(* IEC 61131-3 sources: Automation-Studio-Files/, 2 files *)

(* ---- Global.var ---- *)
VAR
	BtnStart : BOOL;
	BtnStop : BOOL;
	BtnEmStop : BOOL;
	MotorConveyor : BOOL;
	MotorConveyorReverse : BOOL;
END_VAR

(* ---- Main.st ---- *)
PROGRAM _INIT
	(* Insert code here *)

	//BtnStart : BOOL;
//	BtnStop : BOOL;
	//MotorConveyor : BOOL;

END_PROGRAM

PROGRAM _CYCLIC
	(* Insert code here *)

	IF BtnStart THEN
		MotorConveyor := TRUE;
	ELSIF BtnStop THEN
		MotorConveyor := FALSE;
	END_IF

END_PROGRAM

PROGRAM _EXIT
	(* Insert code here *)
	PulleySystem := TRUE ;
//	IF BtnStop THEN
	//	MotorConveyor := FALSE;
//	END_IF

END_PROGRAM
